FUNCTION_BLOCK FB_SystemTimeService
VAR_INPUT
END_VAR
VAR_OUTPUT
END_VAR
VAR
    fbSystemTime    : FB_LocalSystemTime;
    sFileTimeString : STRING;
END_VAR


fbSystemTime(
	sNetID := '',
	bEnable := TRUE,
	dwCycle := 1,
	dwOpt := 0,
	tTimeout := DEFAULT_ADS_TIMEOUT
);

CalculateFileTimeString();

METHOD PRIVATE CalculateFileTimeString : BOOL
VAR_INPUT
END_VAR
VAR
    srawString      : STRING;
    sDeletedString  : STRING;
    sDeletedString2 : STRING;
END_VAR

srawString := ToString;

FindAndDeleteChar( ADR( srawString ), '-', ADR( sDeletedString ), SIZEOF( sDeletedString ) );
FindAndDeleteChar( ADR( sDeletedString ), ':', ADR( sDeletedString2 ), SIZEOF( sDeletedString2 ) );

sFileTimeSTring := Concat( Insert( LEFT( sDeletedString2, LEN( sDeletedString2 ) - 4 ), '_', 8 ), '_' );
END_METHOD

PROPERTY PUBLIC DateTime : DT
GET
DateTime := SYSTEMTIME_TO_DT( fbSystemTime.systemTime );
END_GET
END_PROPERTY

PROPERTY PUBLIC IsValid : BOOL
GET
IsValid := fbSystemTime.bValid;
END_GET
END_PROPERTY

PROPERTY PUBLIC TimeOfDay : TOD
GET
TimeOfDay := DT_TO_TOD( DateTime );
END_GET
END_PROPERTY

PROPERTY TimeOfDayToString : STRING
GET
TimeOfDayToString := RIGHT( ToString, 12 );
END_GET
END_PROPERTY

PROPERTY PUBLIC TimeStruct : REFERENCE TO TIMESTRUCT
GET
TimeStruct REF= fbSystemTime.systemTime;
END_GET
END_PROPERTY

PROPERTY PUBLIC ToFileTimeString : STRING
GET
ToFileTimeString := sFileTimeString;
END_GET
END_PROPERTY

PROPERTY ToString : STRING
GET
ToString := SYSTEMTIME_TO_STRING( fbSystemTime.systemTime );
END_GET
END_PROPERTY

END_FUNCTION_BLOCK

(* stored: Version 1.1.0.1, ProductVersion 3.1.4026.18
   POU FB_SystemTimeService: Id {e7be0e53-d4cf-444b-86b4-b19d0caa481a}, SpecialFunc None
   Method CalculateFileTimeString: Id {4926ae19-31cd-40b3-9d70-7237a41f6da2}
   Property DateTime: Id {18d8d57b-73ed-42f4-8613-1226d7cadce5}
   Get Get: Id {66cc222c-84be-4d38-aba5-734c1286d56d}
   Property IsValid: Id {19272b67-0e7a-411e-8093-227ed218e72a}
   Get Get: Id {df610bc6-de53-4146-9d82-ae04412c3296}
   Property TimeOfDay: Id {341a2e55-ac4e-4e11-936d-734c2dba4e5c}
   Get Get: Id {76a20bbb-63d6-4611-8b37-adbed6704caa}
   Property TimeOfDayToString: Id {22839646-4128-4bcc-a8c2-7fe1015fb5dc}
   Get Get: Id {af561fbb-d828-44d4-91b0-7fc3a6e59850}
   Property TimeStruct: Id {3f05f829-eb00-43eb-8f91-db7068b1653e}
   Get Get: Id {28d18ddc-6cbe-4491-95e2-5984bd4cf324}
   Property ToFileTimeString: Id {e71fa7ac-d773-433c-9504-3e670c55fe56}
   Get Get: Id {900518f2-afd8-4a49-a87c-dfd50b1defcd}
   Property ToString: Id {a4509292-3346-48ce-a241-74c0108a2bf4}
   Get Get: Id {7af9a5ec-e140-4e9b-9e3a-0068a40211ac} *)
